INTERFACE I_Motor

METHOD PUBLIC Start
VAR_INPUT
END_VAR
END_METHOD

METHOD PUBLIC stop : BOOL
VAR_INPUT
END_VAR
END_METHOD

END_INTERFACE

(* stored: Version 1.1.0.1, ProductVersion 3.1.4024.12
   Itf I_Motor: Id {61e3bf94-ecc0-4922-b4e0-8e1daa75e76e}
   Method Start: Id {7cfc481a-0648-4fee-a315-b84f567ad5c1}
   Method stop: Id {a82200c6-31a8-4f6f-be39-375799d996e8} *)
